FUNCTION_BLOCK PKP_2200_LI_4_DI (* Service Interface Function Block Type *)
  (* Standard: SAE J1939; Function: Combo Block: 8 Inputs/8 Outputs (includes all input/output types); Type: DP-34044-1-000; Description: this maps to IX/QX *)
  (* Version 1.0, 2018-12-05, Jose Cabral *)
  (* Version 1.1, 2022-08-04, Franz Hoepfinger, HR Agrartechnik GmbH *)
  (* Version 1.2, 2023-01-05, Franz Hoepfinger, HR Agrartechnik GmbH *)
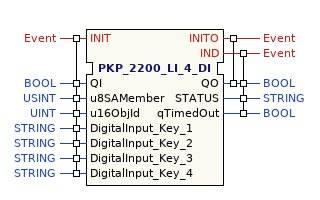
  EVENT_INPUT
    INIT WITH QI, u8SAMember, u16ObjId, DigitalInput_Key_1, DigitalInput_Key_2, DigitalInput_Key_3, DigitalInput_Key_4; (* Service Initialization *)
  END_EVENT
  EVENT_OUTPUT
    INITO WITH QO; (* Initialization Confirm *)
    IND WITH QO, STATUS, qTimedOut; (* Indication from Resource *)
  END_EVENT
  VAR_INPUT
    QI : BOOL; (* Event Input Qualifier *)
    u8SAMember : USINT := PKP_2200_DEFAULT; (* Node SA (Default 21h = PKP_2200_DEFAULT) *)
    u16ObjId : UINT := ID_NULL; (* Dummy ! set to ID_NULL if in Doubt. ID_OFF deactivates FB. *)
    DigitalInput_Key_1 : STRING;
    DigitalInput_Key_2 : STRING;
    DigitalInput_Key_3 : STRING;
    DigitalInput_Key_4 : STRING;
  END_VAR
  VAR_OUTPUT
    QO : BOOL; (* Event Output Qualifier *)
    STATUS : STRING; (* Service Status *)
    qTimedOut : BOOL;
  END_VAR
END_FUNCTION_BLOCK
